TYPE ProfilerStackStruct :
STRUCT
  hash : UINT;
  depth : DINT;
  startlo : LWORD;
  starthi : LWORD;  
  endlo : LWORD;
  endhi : LWORD;  
END_STRUCT
END_TYPE

(* stored: Version 1.1.0.1, ProductVersion 3.1.4020.12
   DUT ProfilerStackStruct: Id {72c79013-bc38-4419-a5a6-7aa37877a660} *)
